FUNCTION_BLOCK E_REND (* Rendezvous (AND) of two events *)
  (* Standard: 61499-1 Annex A; Description: Copyright (c) 2017 fortiss GmbH This program and the accompanying materials are made available under the terms of the Eclipse Public License 2.0 which is available at https://www.eclipse.org/legal/epl-2.0/ SPDX-License-Identifier: EPL-2.0 *)
  (* Version 3.0, 2025-04-14, Patrick Aigner, changed package *)
  (* Version 1.0, 2017-09-20, Alois Zoitl, fortiss GmbH, initial API and implementation and/or initial documentation *)
  PACKAGE iec61499::events;
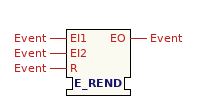
  EVENT_INPUT
    EI1; (* first event to wait for *)
    EI2; (* second event to wait for *)
    R; (* reset the FB to inital state (i.e., wait again for both events) *)
  END_EVENT
  EVENT_OUTPUT
    EO; (* triggered when both EI1 and EI2 occured at least once *)
  END_EVENT
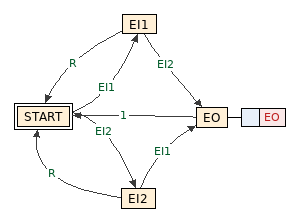
  EC_STATES
    START; (* Initial State *)
    EI1; (* EI1 occured at least once *)
    EO : -> EO; (* Both input events occured at least once send output event *)
    EI2; (* EI2 occured at least once *)
  END_STATES
  EC_TRANSITIONS
    START TO EI2 := EI2;
    START TO EI1 := EI1;
    EI2 TO START := R;
    EI1 TO START := R;
    EI1 TO EO := EI2;
    EI2 TO EO := EI1;
    EO TO START := 1;
  END_TRANSITIONS
END_FUNCTION_BLOCK
